Fanuc KAREL source: kd00009.KL

-- PROVISIONAL review KL for V770-1; original PC SHA256 3edf50d6ca598b2c224dbf64674c308eb87fe643a6dfe1ec049b409c9492c87d
-- Incomplete behavior may be omitted. Consult companion uncertainty JSON. Do not deploy.
PROGRAM KD00009
%NOLOCKGROUP
VAR
  I : INTEGER
  J : INTEGER
  B : BOOLEAN
  R : REAL
  S : STRING[80]
BEGIN
  -- UNRESOLVED_PC offsets 5-12; opcodes 9D,23
  -- UNRESOLVED_PC offsets 17-21; opcodes 7F
END KD00009
